// TIA Portal project "Filling Tank" (V16)
// Vorlageprojekt für das Buch mit Zielsystem S7-1200

(* hardware
DEVICE "S7-1200-Station_1"  S7-1200 Station
   slot 0: "Baugruppenträger_0"  Rack  V1.0
   slot 1: "PLC_1"  CPU 1211C DC/DC/DC  6ES7 211-1AE40-0XB0  V4.1
*)

// ===== PLC "PLC_1"  CPU 1211C DC/DC/DC =====

VAR_GLOBAL   // PLC tag table "Standard-Variablentabelle"
   "fill valve" AT %A0.0 : Bool;
   "FILL" AT %E0.0 : Bool;
   "Discharge" AT %E0.1 : Bool;
   "Tag_4" AT %I10.0 : Bool;
   "Tag_5" AT %Q10.0 : Bool;
   "Tag_6" AT %I10.1 : Bool;
   "Tag_1" AT %M0.0 : Bool;
   "Discharge Valve" AT %Q0.1 : Bool;
   "Tag_2" AT %M0.1 : Bool;
   "Tag_3" AT %QD10 : Time;
   "Tag_7" AT %M1.0 : Bool;
   "Tag_8" AT %M1.1 : Bool;
   "Tag_9" AT %Q0.2 : Bool;
   "Tag_10" AT %Q0.3 : Bool;
   "Tag_11" AT %QD14 : Time;
   "Tag_12" AT %QD22 : Time;
END_VAR

// folder: System blocks/Program resources

DATA_BLOCK "T1"   // DB1
{ S7_Optimized_Access := 'TRUE' }
AUTHOR : Simatic
FAMILY : IEC
NAME : IEC_TMR
VERSION : 1.0
// stored: InstanceOfName IEC_TIMER
"IEC_TIMER"
BEGIN
END_DATA_BLOCK

DATA_BLOCK "T2"   // DB2
{ S7_Optimized_Access := 'TRUE' }
AUTHOR : Simatic
FAMILY : IEC
NAME : IEC_TMR
VERSION : 1.0
// stored: InstanceOfName IEC_TIMER
"IEC_TIMER"
BEGIN
END_DATA_BLOCK

// folder: (top level)

FUNCTION "MHJ-PLC-Lab-Function-S71200" : Void   // FC9000, SCL
{ S7_Optimized_Access := 'TRUE' }
VERSION : 0.1
   VAR_TEMP
      rdTimeReturn : Int;
      outputTime : DTL;
      SyncVal : Byte;
      forVal : Int;
      forVal_2 : Int;
      Value : Byte;
   END_VAR
   VAR CONSTANT
      CompVal : Byte := 16#34;
      Value_01 : Byte := 16#11;
      Value_01_DW : DWord := 16#A165_D992;
      Value_02_DW : DWord := 16#58BE_4401;
   END_VAR
BEGIN

   #Value:=PEEK(area := 16#82,
        dbNumber := 0,
        byteOffset := 511);
   #Value := #Value + 1;

   POKE(area := 16#82,
        dbNumber := 0,
        byteOffset := 511,
        value := #Value);

   POKE(area:=16#81,
        dbNumber:=0,
        byteOffset:=1016,
        value:=#Value_01_DW);
   POKE(area := 16#81,
        dbNumber := 0,
        byteOffset := 1020,
        value := #Value_02_DW);

   POKE(area := 16#81,
        dbNumber := 0,
        byteOffset := 511,
        value := B#16#00);

   FOR #forVal := 0 TO 120 DO
       FOR #forVal_2:=0 TO 10 DO
           #rdTimeReturn:=RD_SYS_T(#outputTime);
           #rdTimeReturn := WR_SYS_T(#outputTime);
           #rdTimeReturn := RD_SYS_T(#outputTime);
           #rdTimeReturn := WR_SYS_T(#outputTime);
       END_FOR;
       #SyncVal:= PEEK(area := 16#81,
                      dbNumber := 0,
                      byteOffset := 511);
       IF #SyncVal = #CompVal THEN
          GOTO M_1;
       END_IF;
   END_FOR;
   RETURN;

   M_1:
   POKE(area := 16#81,
        dbNumber := 0,
        byteOffset := 511,
        value := B#16#0);
END_FUNCTION

ORGANIZATION_BLOCK "Main"   // OB1, LAD, ProgramCycle
TITLE = "Main Program Sweep (Cycle)"
{ S7_Optimized_Access := 'TRUE' }
VERSION : 0.1
   VAR_INPUT
      Initial_Call : Bool;   // Initial call of this OB
      Remanence : Bool;   // =True, if remanent data are available
   END_VAR
BEGIN

REGION Network 1: Konnektierungsbaustein für PLC-Lab
   // Im Netzwerk 1 wird der Konnektierungsbaustein für PLC-Lab aufgerufen.
   // Dieser Aufruf darf nicht entfernt werden!
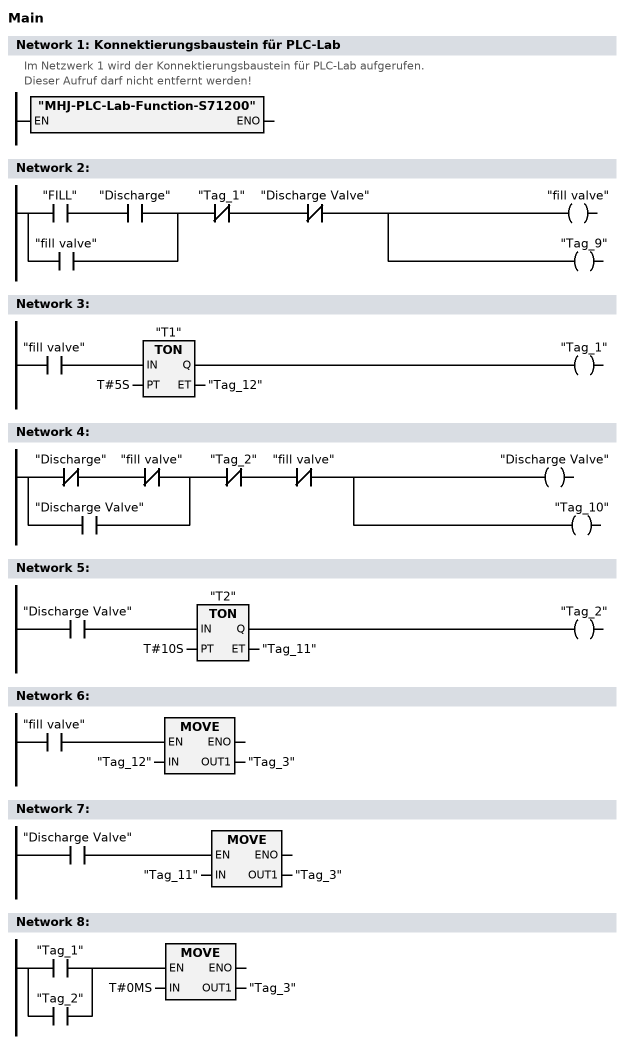
   RUNG wire#powerrail
      "MHJ-PLC-Lab-Function-S71200"()
   END_RUNG
   // the same network as SCL:
   "MHJ-PLC-Lab-Function-S71200"();
END_REGION

REGION Network 2
   RUNG wire#powerrail
      Contact( "FILL" )
      Contact( "Discharge" )
      wire#w1
      I_Contact( "Tag_1" )
      I_Contact( "Discharge Valve" )
      wire#w2
      Coil( "fill valve" )
   END_RUNG
   RUNG wire#powerrail
      Contact( "fill valve" )
   END_RUNG wire#w1
   RUNG wire#w2
      Coil( "Tag_9" )
   END_RUNG
   // the same network as SCL:
   "fill valve" := (("FILL" AND "Discharge") OR "fill valve") AND NOT "Tag_1" AND NOT "Discharge Valve";
   "Tag_9" := "fill valve";
END_REGION

REGION Network 3
   "T1".TON(IN := "fill valve", PT := T#5S, ET => "Tag_12");
   "Tag_1" := "T1".Q;
END_REGION

REGION Network 4
   RUNG wire#powerrail
      I_Contact( "Discharge" )
      I_Contact( "fill valve" )
      wire#w1
      I_Contact( "Tag_2" )
      I_Contact( "fill valve" )
      wire#w2
      Coil( "Discharge Valve" )
   END_RUNG
   RUNG wire#powerrail
      Contact( "Discharge Valve" )
   END_RUNG wire#w1
   RUNG wire#w2
      Coil( "Tag_10" )
   END_RUNG
   // the same network as SCL:
   "Discharge Valve" := ((NOT "Discharge" AND NOT "fill valve") OR "Discharge Valve") AND NOT "Tag_2" AND NOT "fill valve";
   "Tag_10" := "Discharge Valve";
END_REGION

REGION Network 5
   "T2".TON(IN := "Discharge Valve", PT := T#10S, ET => "Tag_11");
   "Tag_2" := "T2".Q;
END_REGION

REGION Network 6
   RUNG wire#powerrail
      Contact( "fill valve" )
      Move(in := "Tag_12", out1 => "Tag_3")
   END_RUNG
   // the same network as SCL:
   IF "fill valve" THEN "Tag_3" := "Tag_12"; END_IF;
END_REGION

REGION Network 7
   RUNG wire#powerrail
      Contact( "Discharge Valve" )
      Move(in := "Tag_11", out1 => "Tag_3")
   END_RUNG
   // the same network as SCL:
   IF "Discharge Valve" THEN "Tag_3" := "Tag_11"; END_IF;
END_REGION

REGION Network 8
   RUNG wire#powerrail
      Contact( "Tag_1" )
      wire#w1
      Move(in := T#0MS, out1 => "Tag_3")
   END_RUNG
   RUNG wire#powerrail
      Contact( "Tag_2" )
   END_RUNG wire#w1
   // the same network as SCL:
   IF "Tag_1" OR "Tag_2" THEN "Tag_3" := T#0MS; END_IF;
END_REGION
END_ORGANIZATION_BLOCK